Omron CX-Programmer project NewProject (CX-Programmer 9.75)

# PLC project03: CP2E-N N

## Program NewProgram1 (cyclic task 0)

### Section Section1

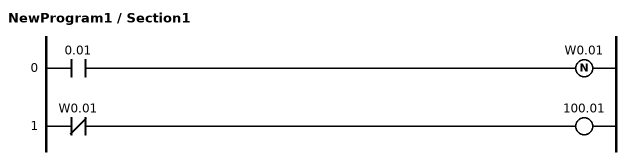
; rung 0
LD 0.01
DIFD(014) W0.01
; rung 1
LDNOT W0.01
OUT 100.01

### Section END
; rung 0
END(001)